# EPICS StreamDevice protocol: iocs/rpi-cherenkov/cherenkov_serial.proto
Terminator = CR LF;

ReadTimeout = 1000;
#WriteTimeout = 100;
#PollPeriod = 400;

ExtraInput = Ignore;

# serial device returns the adc values as long data type. Also the values are in micro volts

read_CH0 {
#	out "CH1";
	in "0CH%i";
}

read_CH1 {
#	out "CH2";
	in "1CH%i";
}

read_CH2 {
#	out "CH3";
	in "2CH%i";
}

read_CH3 {
#	out "CH4";
	in "3CH%i";
}
